FUNCTION_BLOCK StringBuilder IMPLEMENTS IStringBuilder, ILimitedStringBuilder
VAR_INPUT
END_VAR
VAR_OUTPUT
END_VAR
VAR
	{attribute 'hide'}
    _workString : STRING;
END_VAR

METHOD Append : IStringBuilder
VAR_INPUT
    text : STRING; 
END_VAR
_workString := CONCAT(_workString, text);
Append := THIS^;
END_METHOD

METHOD InsertAtLocation : REFERENCE TO StringBuilder
VAR_INPUT
    Text : STRING;
    Position : INT;
END_VAR
_workString := Tc2_Standard.INSERT(_WorkString, Text, Position);
InsertAtLocation REF= THIS^;
END_METHOD

METHOD Reset : ILimitedStringBuilder
_workString := '';
Reset := THIS^;
END_METHOD

METHOD ToString : STRING
ToString := _workString;
END_METHOD

END_FUNCTION_BLOCK

(* stored: Version 1.1.0.1, ProductVersion 3.1.4024.3
   POU StringBuilder: Id {cb83af3e-7acc-470f-a3f2-ea518b91b0ac}, SpecialFunc None
   Method Append: Id {eb17deb0-cac2-49f1-9f9e-8c5927d682db}
   Method InsertAtLocation: Id {62589235-1008-41ba-bd68-cb90dfa17d3b}
   Method Reset: Id {7fc6d06f-fa1c-475b-830c-8199514fa190}
   Method ToString: Id {d9afa94d-09f4-4404-8482-75a4b3c27ac8} *)
